Staubli VAL3: getX.pgx

public program getX(num& nValueX (dimensions=1))
  local point pHere
begin
  pHere=here(tActive,frActive)
  nValueX=pHere.trsf.x
end
